DATA_BLOCK "ST10_Flow7_CGlueing_iDB"
{ S7_Optimized_Access := 'TRUE' }
VERSION : 0.1
NON_RETAIN
"ST10_Flow7_CGlueing"

BEGIN

END_DATA_BLOCK

